// TIA Portal V19 export
TYPE "type_materialParError"
// stored: Access Published
   STRUCT
      error : Bool;   // Manual mode parameters for axis control interface
   END_STRUCT;
END_TYPE
